PROGRAM MAIN

(* ========================================================= *)
(*    PRG: TwinCAT CNC                                       *)
(* --------------------------------------------------------- *)
(*  Desc: Base PLC program for TwinCAT CNC                  *)
(* 	Author: MK                                                *)
(*  Date: 21.12.2011                                        *)
(*  Cust.:                                                   *)
(*  M-No:                                                   *)
(*  Kom.:                                                   *)
(*  Rev.: 1.3  from 1.24                                    *)
(* ========================================================= *)

DemoSine();
DemoUpDown();
DemoTest();
WritePersistentData();
ShowMessages();
MySystemTime();

HLI_Init();
IF CncSystem.bHLIInit = TRUE THEN
	CncPlcProgram();
	CncMFunctions();
	CncPlcManualFunctions();
	CncPlcMessages();
	CncRefPosOffs();
	CncVariables();
	CncHmiData();
	
	//gpAx[0]^.ipo_mc_control.emergency_stop.command_w :=1;
	
	//Axis1CurrPosition := gpAx[0]^.lr_state.current_position_acs_r/10000.0;
	//Axis2CurrPosition := gpAx[0]^.lr_state.current_position_acs_r/10000.0;
	//Axis3CurrPosition := gpAx[0]^.lr_state.current_position_acs_r/10000.0;
	
END_IF



								(*--Belo Controlador--*)
TController_Enable();
								
								(* -- Set das variáveis para a HMI -- *)
SetHMIVariables();

END_PROGRAM

(* stored: Version 1.1.0.1, ProductVersion 3.1.4020.12
   POU MAIN: Id {56a94792-f833-4bc1-a3f7-6ceccad4dcc0}, SpecialFunc None *)
